TYPE ST_TOLERANCETHRESHOLDPK :
STRUCT
	GOODREADPERCENTAGECS	:STRING;
	GOODREADPERCENTAGEOUT	:STRING;
END_STRUCT
END_TYPE

(* stored: Version 1.1.0.1, ProductVersion 3.1.4024.13
   DUT ST_TOLERANCETHRESHOLDPK: Id {1d17263f-4f75-4a77-938e-3dbb4ec5ea2e} *)
